(* PLC project canopen_slave, lolitech beremiz 1 *)
(* stored: creationDateTime 2008-06-24T18:44:00, modificationDateTime 2008-10-24T09:32:01, language en-US *)

PROGRAM test_main
  VAR
    outvar AT %QW0.0.8192.0 : INT;
    invar AT %IW0.0.8193.0 : INT;
  END_VAR

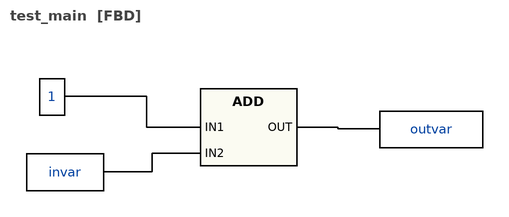
(* FBD diagram, written out as Structured Text *)
outvar := 1 + invar;
END_PROGRAM

CONFIGURATION conf
  RESOURCE res ON PLC
    TASK tache(INTERVAL := 00:00:00.010000, PRIORITY := 0);
    PROGRAM toto WITH tache : test_main;
  END_RESOURCE
END_CONFIGURATION
